PROGRAM MAIN
VAR
	bActivateMotion : BOOL;
	fVelRef : LREAL;
	fPosRef : LREAL;
	fPodMeas : LREAL;




END_VAR

// Comment out as needed

HMISimulation();
//CraneSteering();

// Ka er Qmax? Til FB_openloopcontrol

END_PROGRAM

(* stored: Version 1.1.0.1, ProductVersion 3.1.4024.10
   POU MAIN: Id {0ad4954e-ac64-46bb-9eb0-a0f0715ea3b1}, SpecialFunc None *)
